PROGRAM Example04_2DoFs_Synchronized_Waypoints_2
VAR
  otg : Ruckig(0.001, 2) := (Synchronization := SynchronizationType.TimeSync,
                               MaxVelocity :=         [ 10.0, 10.0 ],
                               MaxAcceleration :=     [ 50000.0, 50000.0 ],
                               MaxJerk :=             [ 500000.0, 500000.0 ],
                               CurrentPosition :=     [ 0.0, 0.0 ],
                               CurrentVelocity :=     [ 0.0, 0.0 ],
                               CurrentAcceleration := [ 0.0, 0.0 ],
                               TargetPosition :=      [ 0.0, 0.0 ],
                               TargetVelocity :=      [ 0.0, 0.0 ],
                               TargetAcceleration :=  [ 0.0, 0.0 ]);							   
  waypoints : INT := 50;
  a : LREAL := 300;
  b : LREAL := 200;
  w1 : LREAL := 3;
  w2 : LREAL := 2;
  delta : LREAL := PI * 0.5;
  currentWaypoint : INT := 0;
  firstRun : BOOL := TRUE;
  dump : LREAL; // just for testing
END_VAR

// init trajectory
IF firstRun
THEN
  firstRun := FALSE;
  Waypoint(currentWaypoint, px := otg.CurrentPosition[0], py := otg.CurrentPosition[1],
                            vx := otg.CurrentVelocity[0], 
                            vy := otg.CurrentVelocity[1],
                            ax := otg.CurrentAcceleration[0], 
                            ay := otg.CurrentAcceleration[1]
							);
  otg.TargetPosition := otg.CurrentPosition;
  otg.TargetVelocity := otg.CurrentVelocity;
  otg.TargetAcceleration := otg.CurrentAcceleration;  
END_IF

// increment waypoints
otg(EnableAutoPropagate := TRUE);
IF otg.State = TrajectoryState.Idle
THEN
  Waypoint(currentWaypoint, px := otg.TargetPosition[0], py := otg.TargetPosition[1],
                            vx := otg.TargetVelocity[0], 
                            vy := otg.TargetVelocity[1],
                            ax := dump, //otg.Input.TargetAcceleration[0], 
                            ay := dump //otg.Input.TargetAcceleration[1]);
							);
  currentWaypoint := SEL(currentWaypoint + 1 < waypoints, 0, currentWaypoint+1);
END_IF

METHOD Waypoint
VAR_INPUT
  w : INT;
END_VAR
VAR_IN_OUT
  px, py : LREAL;
  vx, vy : LREAL;
  ax, ay : LREAL;
END_VAR
VAR
  offsetx : LREAL;
END_VAR
offsetx := 10 * TRUNC(ABS(w-1)/2);
w := w MOD 2;
CASE w
OF
  0:
    px := offsetx; py := 0;
    vx := 0; vy := 0;
    ax := 0; ay := 0;
  1:
    px := 100 + offsetx; py := 10;
    vx := 0; vy := 0;
    ax := 0; ay := 0;
END_CASE
END_METHOD

END_PROGRAM

(* stored: Version 1.1.0.1, ProductVersion 3.1.4024.9
   POU Example04_2DoFs_Synchronized_Waypoints_2: Id {130c9296-914b-47cf-a456-2f87beca5147}, SpecialFunc None
   Method Waypoint: Id {d23aed48-98fa-4e0a-8baa-7c4cbff31b88} *)
